// TIA Portal V20 export
DATA_BLOCK "HmiInterface"   // DB99
// stored: Access Published, MemoryReserve 100, Namespace Unit1.Em4
   VAR
      em : "LAF_typeEmInterface";
      emHomedCheck : "Unit1.Em4.typeEmHomedCheck";
      cm : "Unit1.Em4.typeCmInterface";
      cutter : "LER_typeSequenceInterface";
   END_VAR
   VAR RETAIN
      cmCompensatorAxisZ : "LBC_typeAxisControlInterface";
      cmFeedingRollAxisB : "LBC_typeAxisControlInterface";
      cmElectrodeCutterAxisZ : "LBC_typeAxisControlInterface";
      cmPositionMovingAxisX : "LBC_typeAxis64PosInterface";
      cmFeederCylinderUpDown : "LBC_typeTwoWayActuatorInterface";
      cmCompensatorSafetyPinIdlePosition : "LBC_typeDigitalSignalInterface";
      cmTabDetectSensor : "LBC_typeDigitalSignalInterface";
      cmTapeDetectSensor : "LBC_typeDigitalSignalInterface";
      cmCutterEpcAnalogInput : "LBC_typeAnalogInputInterface";
      cmCompensatorAxisZ_TorqueCal : "LER_typeServoTorqueCalInterface";
      cmFeedingRollAxisB_TorqueCal : "LER_typeServoTorqueCalInterface";
      cmElectrodeCutterAxisZ_TorqueCal : "LER_typeServoTorqueCalInterface";
      cmPositionMovingAxisX_TorqueCal : "LER_typeServoTorqueCalInterface";
      cutterLifeCount : "LER_typeAlarmCounterInterface";
      tabSensorNotDetectedCount : "LER_typeAlarmCounterInterface";
   END_VAR
BEGIN
   cmCutterEpcAnalogInput.configuration.limitHigh2 := 100.0;
END_DATA_BLOCK
